Xinje XDPPro project, PLC1: XD3-32 (software 3.7.14 2021-12-24)

PROGRAM 梯形图

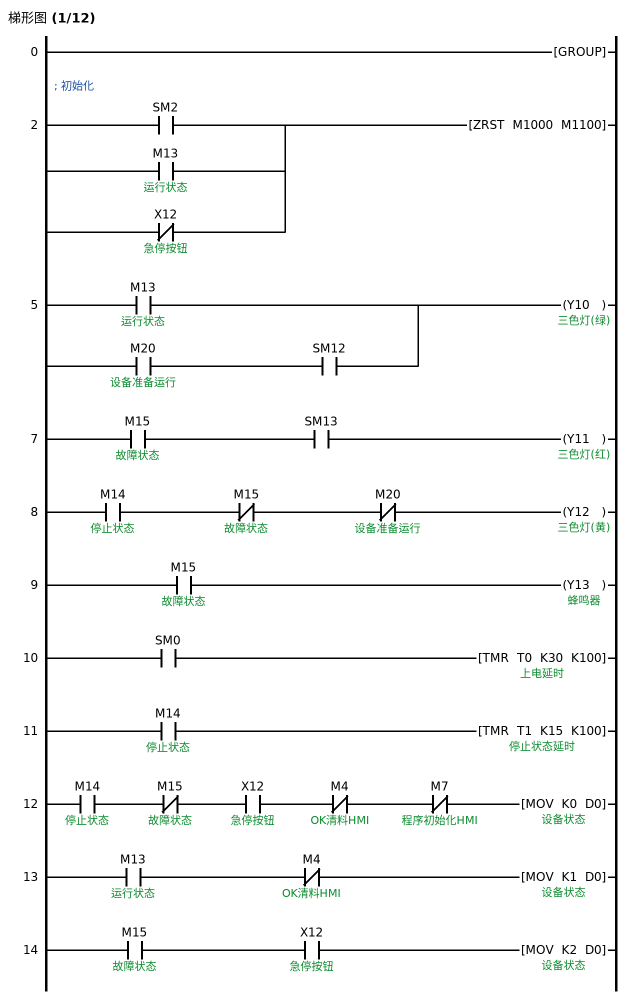
GROUP
; 初始化
LD     SM2
OR     M13	; 运行状态
ORI    X12	; 急停按钮
ZRST   M1000 M1100
LD     M13	; 运行状态
LD     M20	; 设备准备运行
AND    SM12
ORB
OUT    Y10	; 三色灯(绿)
LD     M15	; 故障状态
AND    SM13
OUT    Y11	; 三色灯(红)
LD     M14	; 停止状态
ANI    M15	; 故障状态
ANI    M20	; 设备准备运行
OUT    Y12	; 三色灯(黄)
LD     M15	; 故障状态
OUT    Y13	; 蜂鸣器
LD     SM0
TMR    T0 K30 K100	; 上电延时
LD     M14	; 停止状态
TMR    T1 K15 K100	; 停止状态延时
LD     M14	; 停止状态
ANI    M15	; 故障状态
AND    X12	; 急停按钮
ANI    M4	; OK清料HMI
ANI    M7	; 程序初始化HMI
MOV    K0 D0	; 设备状态
LD     M13	; 运行状态
ANI    M4	; OK清料HMI
MOV    K1 D0	; 设备状态
LD     M15	; 故障状态
AND    X12	; 急停按钮
MOV    K2 D0	; 设备状态

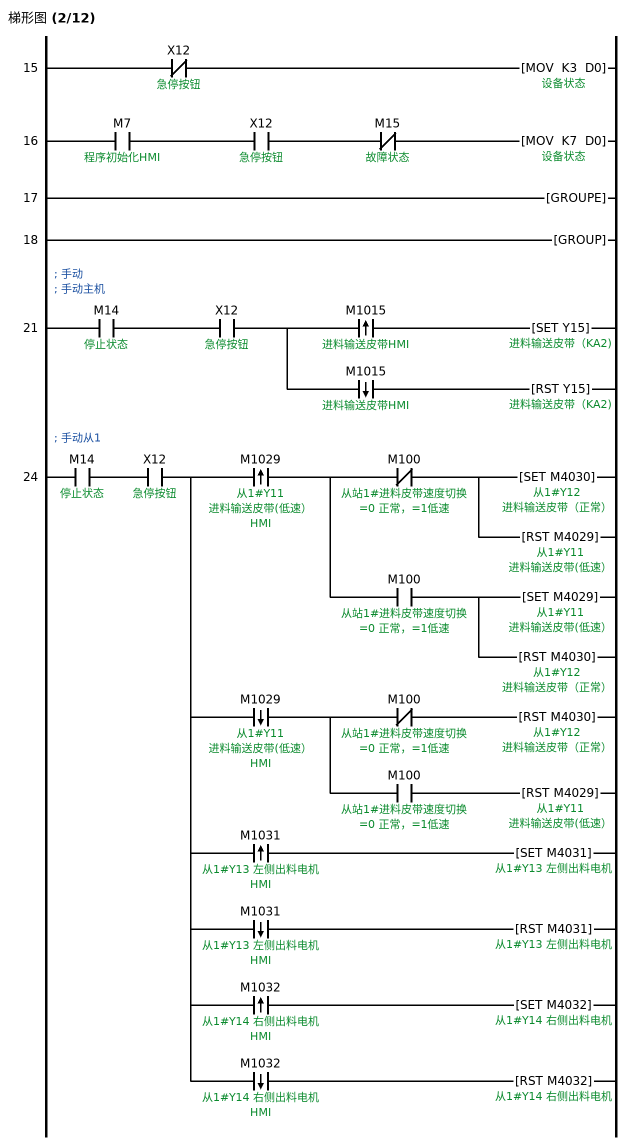
LDI    X12	; 急停按钮
MOV    K3 D0	; 设备状态
LD     M7	; 程序初始化HMI
AND    X12	; 急停按钮
ANI    M15	; 故障状态
MOV    K7 D0	; 设备状态
GROUPE
GROUP
; 手动
; 手动主机
LD     M14	; 停止状态
AND    X12	; 急停按钮
MPS
ANDP   M1015	; 进料输送皮带HMI
SET    Y15	; 进料输送皮带（KA2)
MPP
ANDF   M1015	; 进料输送皮带HMI
RST    Y15	; 进料输送皮带（KA2)
; 手动从1
LD     M14	; 停止状态
AND    X12	; 急停按钮
MPS
ANDP   M1029	; 从1#Y11 进料输送皮带(低速）       HMI
MPS
ANI    M100	; 从站1#进料皮带速度切换=0 正常，=1低速
SET    M4030	; 从1#Y12 进料输送皮带（正常）
RST    M4029	; 从1#Y11 进料输送皮带(低速）
MPP
AND    M100	; 从站1#进料皮带速度切换=0 正常，=1低速
SET    M4029	; 从1#Y11 进料输送皮带(低速）
RST    M4030	; 从1#Y12 进料输送皮带（正常）
MRD
ANDF   M1029	; 从1#Y11 进料输送皮带(低速）       HMI
MPS
ANI    M100	; 从站1#进料皮带速度切换=0 正常，=1低速
RST    M4030	; 从1#Y12 进料输送皮带（正常）
MPP
AND    M100	; 从站1#进料皮带速度切换=0 正常，=1低速
RST    M4029	; 从1#Y11 进料输送皮带(低速）
MRD
ANDP   M1031	; 从1#Y13 左侧出料电机       HMI
SET    M4031	; 从1#Y13 左侧出料电机
MRD
ANDF   M1031	; 从1#Y13 左侧出料电机       HMI
RST    M4031	; 从1#Y13 左侧出料电机
MRD
ANDP   M1032	; 从1#Y14 右侧出料电机       HMI
SET    M4032	; 从1#Y14 右侧出料电机
MPP
ANDF   M1032	; 从1#Y14 右侧出料电机       HMI
RST    M4032	; 从1#Y14 右侧出料电机

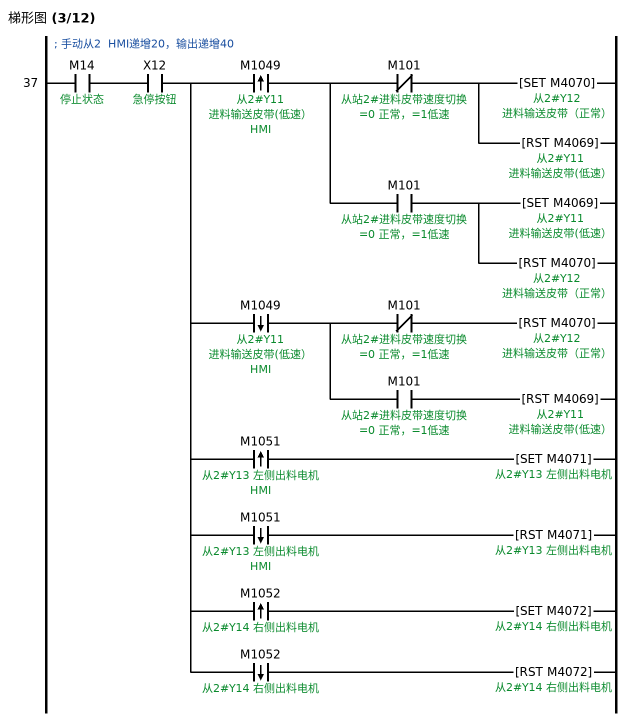
; 手动从2  HMI递增20，输出递增40
LD     M14	; 停止状态
AND    X12	; 急停按钮
MPS
ANDP   M1049	; 从2#Y11 进料输送皮带(低速）       HMI
MPS
ANI    M101	; 从站2#进料皮带速度切换=0 正常，=1低速
SET    M4070	; 从2#Y12 进料输送皮带（正常）
RST    M4069	; 从2#Y11 进料输送皮带(低速）
MPP
AND    M101	; 从站2#进料皮带速度切换=0 正常，=1低速
SET    M4069	; 从2#Y11 进料输送皮带(低速）
RST    M4070	; 从2#Y12 进料输送皮带（正常）
MRD
ANDF   M1049	; 从2#Y11 进料输送皮带(低速）       HMI
MPS
ANI    M101	; 从站2#进料皮带速度切换=0 正常，=1低速
RST    M4070	; 从2#Y12 进料输送皮带（正常）
MPP
AND    M101	; 从站2#进料皮带速度切换=0 正常，=1低速
RST    M4069	; 从2#Y11 进料输送皮带(低速）
MRD
ANDP   M1051	; 从2#Y13 左侧出料电机       HMI
SET    M4071	; 从2#Y13 左侧出料电机
MRD
ANDF   M1051	; 从2#Y13 左侧出料电机       HMI
RST    M4071	; 从2#Y13 左侧出料电机
MRD
ANDP   M1052	; 从2#Y14 右侧出料电机
SET    M4072	; 从2#Y14 右侧出料电机
MPP
ANDF   M1052	; 从2#Y14 右侧出料电机
RST    M4072	; 从2#Y14 右侧出料电机

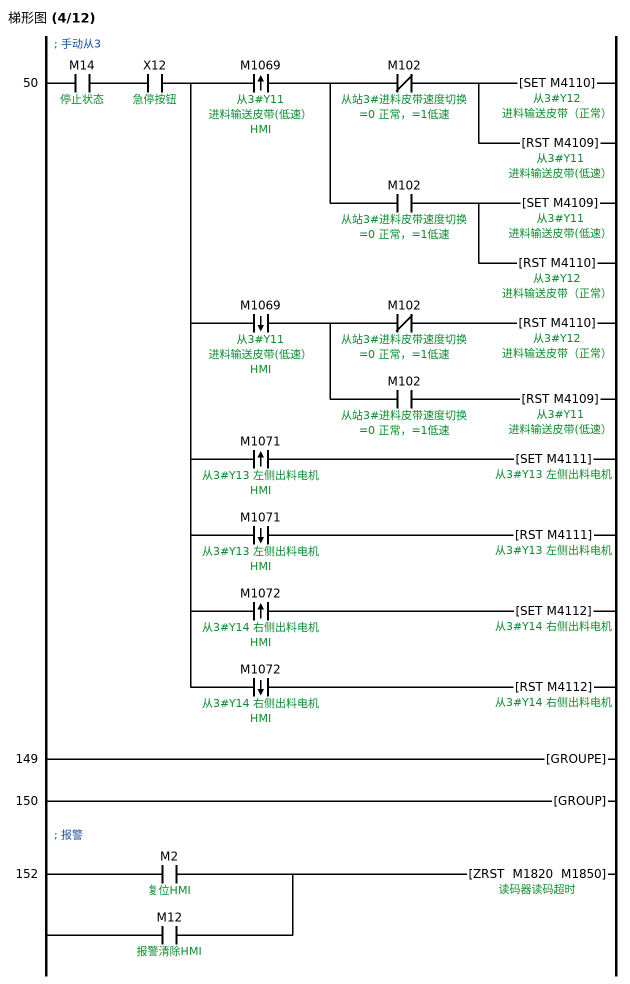
; 手动从3
LD     M14	; 停止状态
AND    X12	; 急停按钮
MPS
ANDP   M1069	; 从3#Y11 进料输送皮带(低速）       HMI
MPS
ANI    M102	; 从站3#进料皮带速度切换=0 正常，=1低速
SET    M4110	; 从3#Y12 进料输送皮带（正常）
RST    M4109	; 从3#Y11 进料输送皮带(低速）
MPP
AND    M102	; 从站3#进料皮带速度切换=0 正常，=1低速
SET    M4109	; 从3#Y11 进料输送皮带(低速）
RST    M4110	; 从3#Y12 进料输送皮带（正常）
MRD
ANDF   M1069	; 从3#Y11 进料输送皮带(低速）       HMI
MPS
ANI    M102	; 从站3#进料皮带速度切换=0 正常，=1低速
RST    M4110	; 从3#Y12 进料输送皮带（正常）
MPP
AND    M102	; 从站3#进料皮带速度切换=0 正常，=1低速
RST    M4109	; 从3#Y11 进料输送皮带(低速）
MRD
ANDP   M1071	; 从3#Y13 左侧出料电机       HMI
SET    M4111	; 从3#Y13 左侧出料电机
MRD
ANDF   M1071	; 从3#Y13 左侧出料电机       HMI
RST    M4111	; 从3#Y13 左侧出料电机
MRD
ANDP   M1072	; 从3#Y14 右侧出料电机       HMI
SET    M4112	; 从3#Y14 右侧出料电机
MPP
ANDF   M1072	; 从3#Y14 右侧出料电机       HMI
RST    M4112	; 从3#Y14 右侧出料电机
GROUPE
GROUP
; 报警
LD     M2	; 复位HMI
OR     M12	; 报警清除HMI
ZRST   M1820 M1850	; 读码器读码超时

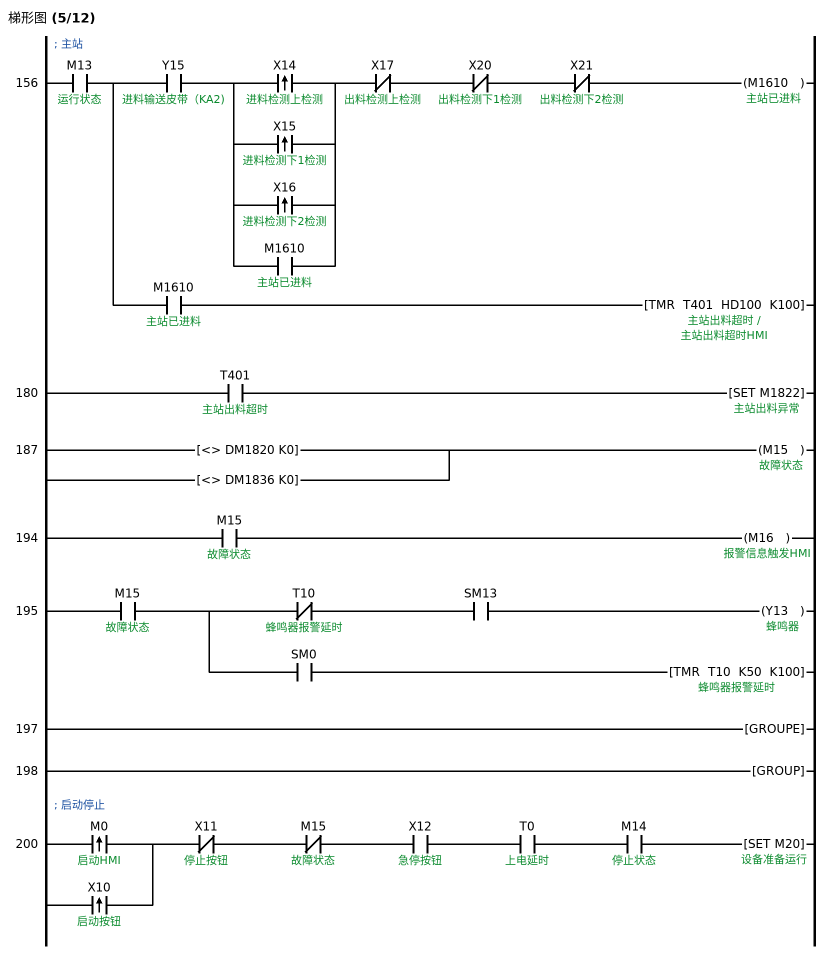
; 主站
LD     M13	; 运行状态
MPS
AND    Y15	; 进料输送皮带（KA2)
LDP    X14	; 进料检测上检测
ORP    X15	; 进料检测下1检测
ORP    X16	; 进料检测下2检测
OR     M1610	; 主站已进料
ANB
ANI    X17	; 出料检测上检测
ANI    X20	; 出料检测下1检测
ANI    X21	; 出料检测下2检测
OUT    M1610	; 主站已进料
MPP
AND    M1610	; 主站已进料
TMR    T401 HD100 K100	; 主站出料超时 / 主站出料超时HMI
LD     T401	; 主站出料超时
SET    M1822	; 主站出料异常
LD<>   DM1820 K0
OR<>   DM1836 K0
OUT    M15	; 故障状态
LD     M15	; 故障状态
OUT    M16	; 报警信息触发HMI
LD     M15	; 故障状态
MPS
ANI    T10	; 蜂鸣器报警延时
AND    SM13
OUT    Y13	; 蜂鸣器
MPP
AND    SM0
TMR    T10 K50 K100	; 蜂鸣器报警延时
GROUPE
GROUP
; 启动停止
LDP    M0	; 启动HMI
ORP    X10	; 启动按钮
ANI    X11	; 停止按钮
ANI    M15	; 故障状态
AND    X12	; 急停按钮
AND    T0	; 上电延时
AND    M14	; 停止状态
SET    M20	; 设备准备运行

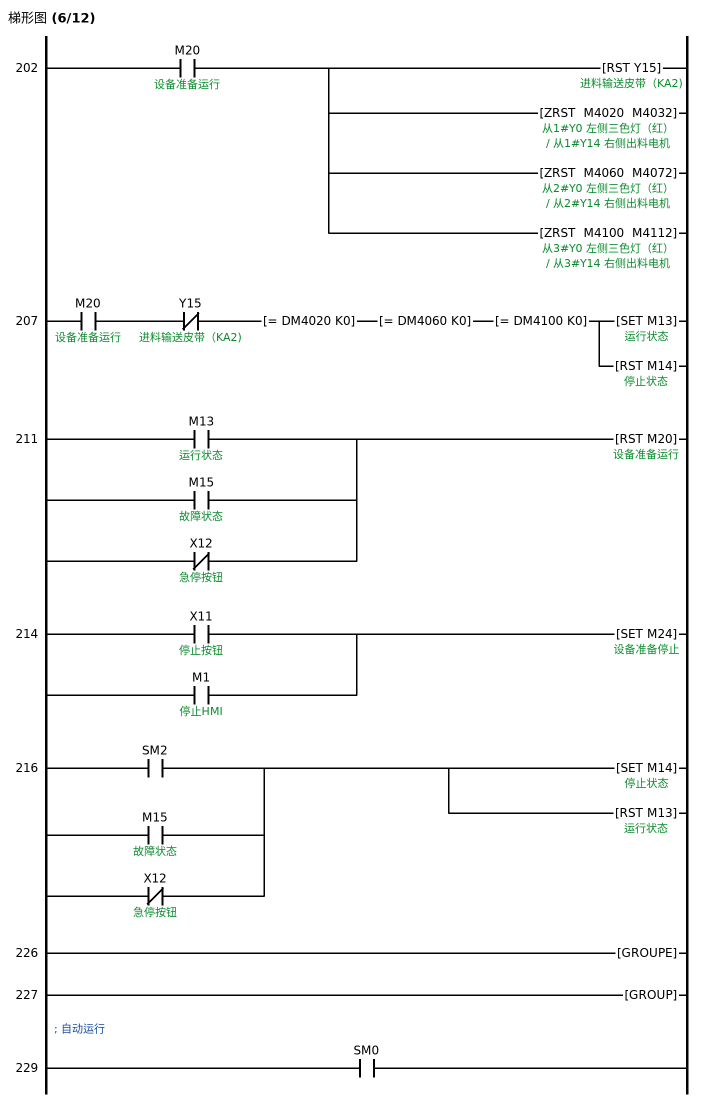
LD     M20	; 设备准备运行
RST    Y15	; 进料输送皮带（KA2)
ZRST   M4020 M4032	; 从1#Y0 左侧三色灯（红） / 从1#Y14 右侧出料电机
ZRST   M4060 M4072	; 从2#Y0 左侧三色灯（红） / 从2#Y14 右侧出料电机
ZRST   M4100 M4112	; 从3#Y0 左侧三色灯（红） / 从3#Y14 右侧出料电机
LD     M20	; 设备准备运行
ANI    Y15	; 进料输送皮带（KA2)
AND=   DM4020 K0
AND=   DM4060 K0
AND=   DM4100 K0
SET    M13	; 运行状态
RST    M14	; 停止状态
LD     M13	; 运行状态
OR     M15	; 故障状态
ORI    X12	; 急停按钮
RST    M20	; 设备准备运行
LD     X11	; 停止按钮
OR     M1	; 停止HMI
SET    M24	; 设备准备停止
LD     SM2
OR     M15	; 故障状态
ORI    X12	; 急停按钮
SET    M14	; 停止状态
RST    M13	; 运行状态
GROUPE
GROUP
; 自动运行
LD     SM0

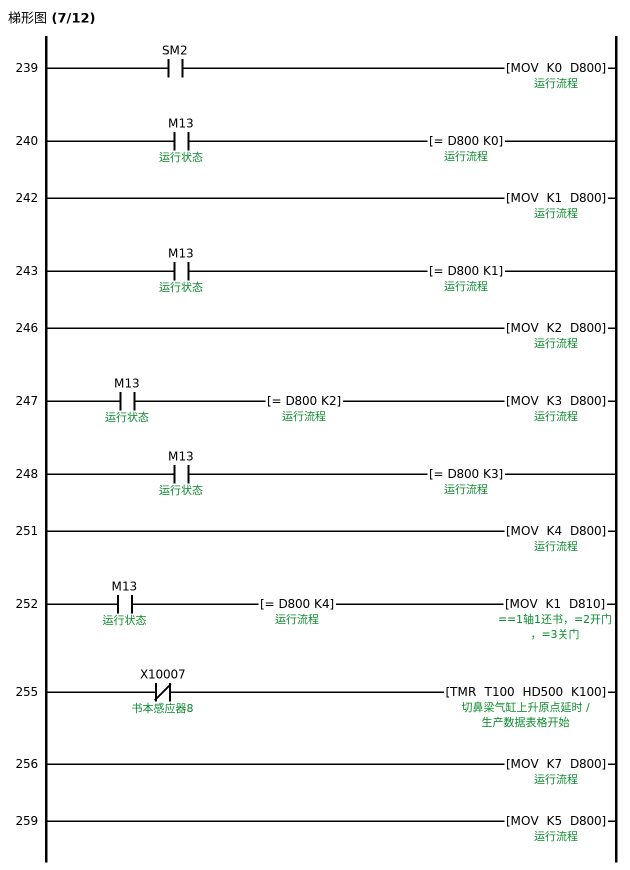
LD     SM2
MOV    K0 D800	; 运行流程
LD     M13	; 运行状态
AND=   D800 K0	; 运行流程
MOV    K1 D800	; 运行流程
LD     M13	; 运行状态
AND=   D800 K1	; 运行流程
MOV    K2 D800	; 运行流程
LD     M13	; 运行状态
AND=   D800 K2	; 运行流程
MOV    K3 D800	; 运行流程
LD     M13	; 运行状态
AND=   D800 K3	; 运行流程
MOV    K4 D800	; 运行流程
LD     M13	; 运行状态
AND=   D800 K4	; 运行流程
MOV    K1 D810	; ==1轴1还书，=2开门，=3关门
LDI    X10007	; 书本感应器8
TMR    T100 HD500 K100	; 切鼻梁气缸上升原点延时 / 生产数据表格开始
MOV    K7 D800	; 运行流程
MOV    K5 D800	; 运行流程

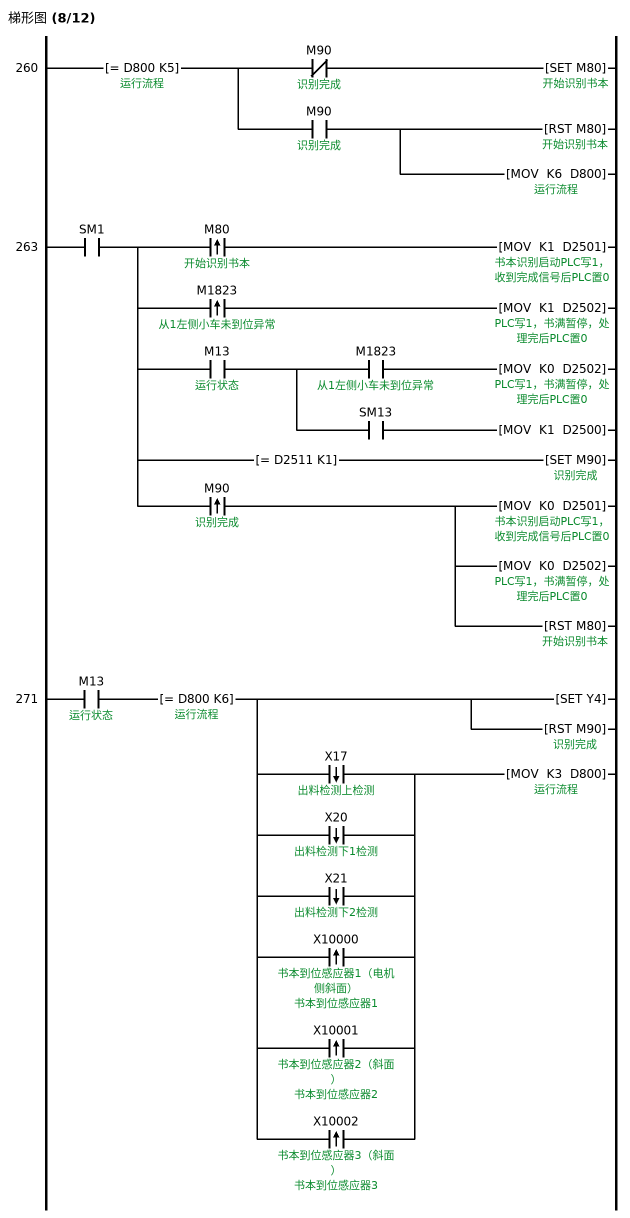
LD=    D800 K5	; 运行流程
MPS
ANI    M90	; 识别完成
SET    M80	; 开始识别书本
MPP
AND    M90	; 识别完成
RST    M80	; 开始识别书本
MOV    K6 D800	; 运行流程
LD     SM1
MPS
ANDP   M80	; 开始识别书本
MOV    K1 D2501	; 书本识别启动PLC写1，收到完成信号后PLC置0
MRD
ANDP   M1823	; 从1左侧小车未到位异常
MOV    K1 D2502	; PLC写1，书满暂停，处理完后PLC置0
MRD
AND    M13	; 运行状态
MPS
AND    M1823	; 从1左侧小车未到位异常
MOV    K0 D2502	; PLC写1，书满暂停，处理完后PLC置0
MPP
AND    SM13
MOV    K1 D2500
MRD
AND=   D2511 K1
SET    M90	; 识别完成
MPP
ANDP   M90	; 识别完成
MOV    K0 D2501	; 书本识别启动PLC写1，收到完成信号后PLC置0
MOV    K0 D2502	; PLC写1，书满暂停，处理完后PLC置0
RST    M80	; 开始识别书本
LD     M13	; 运行状态
AND=   D800 K6	; 运行流程
SET    Y4
RST    M90	; 识别完成
LDF    X17	; 出料检测上检测
ORF    X20	; 出料检测下1检测
ORF    X21	; 出料检测下2检测
ORP    X10000	; 书本到位感应器1（电机侧斜面）       书本到位感应器1
ORP    X10001	; 书本到位感应器2（斜面）             书本到位感应器2
ORP    X10002	; 书本到位感应器3（斜面）             书本到位感应器3
ANB
MOV    K3 D800	; 运行流程

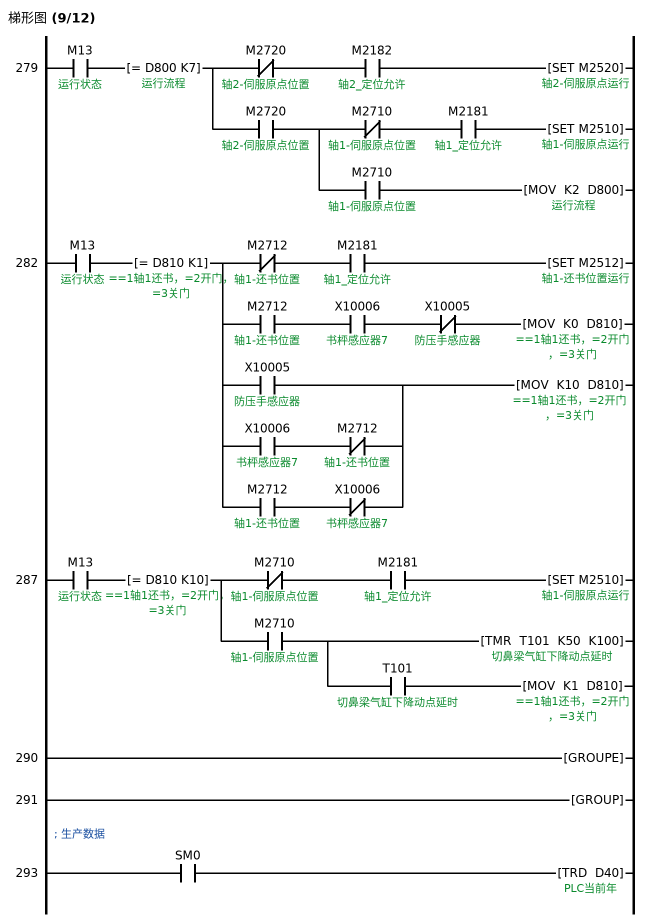
LD     M13	; 运行状态
AND=   D800 K7	; 运行流程
MPS
ANI    M2720	; 轴2-伺服原点位置
AND    M2182	; 轴2_定位允许
SET    M2520	; 轴2-伺服原点运行
MPP
AND    M2720	; 轴2-伺服原点位置
MPS
ANI    M2710	; 轴1-伺服原点位置
AND    M2181	; 轴1_定位允许
SET    M2510	; 轴1-伺服原点运行
MPP
AND    M2710	; 轴1-伺服原点位置
MOV    K2 D800	; 运行流程
LD     M13	; 运行状态
AND=   D810 K1	; ==1轴1还书，=2开门，=3关门
MPS
ANI    M2712	; 轴1-还书位置
AND    M2181	; 轴1_定位允许
SET    M2512	; 轴1-还书位置运行
MRD
AND    M2712	; 轴1-还书位置
AND    X10006	; 书枰感应器7
ANI    X10005	; 防压手感应器
MOV    K0 D810	; ==1轴1还书，=2开门，=3关门
MPP
LD     X10005	; 防压手感应器
LD     X10006	; 书枰感应器7
ANI    M2712	; 轴1-还书位置
ORB
LD     M2712	; 轴1-还书位置
ANI    X10006	; 书枰感应器7
ORB
ANB
MOV    K10 D810	; ==1轴1还书，=2开门，=3关门
LD     M13	; 运行状态
AND=   D810 K10	; ==1轴1还书，=2开门，=3关门
MPS
ANI    M2710	; 轴1-伺服原点位置
AND    M2181	; 轴1_定位允许
SET    M2510	; 轴1-伺服原点运行
MPP
AND    M2710	; 轴1-伺服原点位置
TMR    T101 K50 K100	; 切鼻梁气缸下降动点延时
AND    T101	; 切鼻梁气缸下降动点延时
MOV    K1 D810	; ==1轴1还书，=2开门，=3关门
GROUPE
GROUP
; 生产数据
LD     SM0
TRD    D40	; PLC当前年

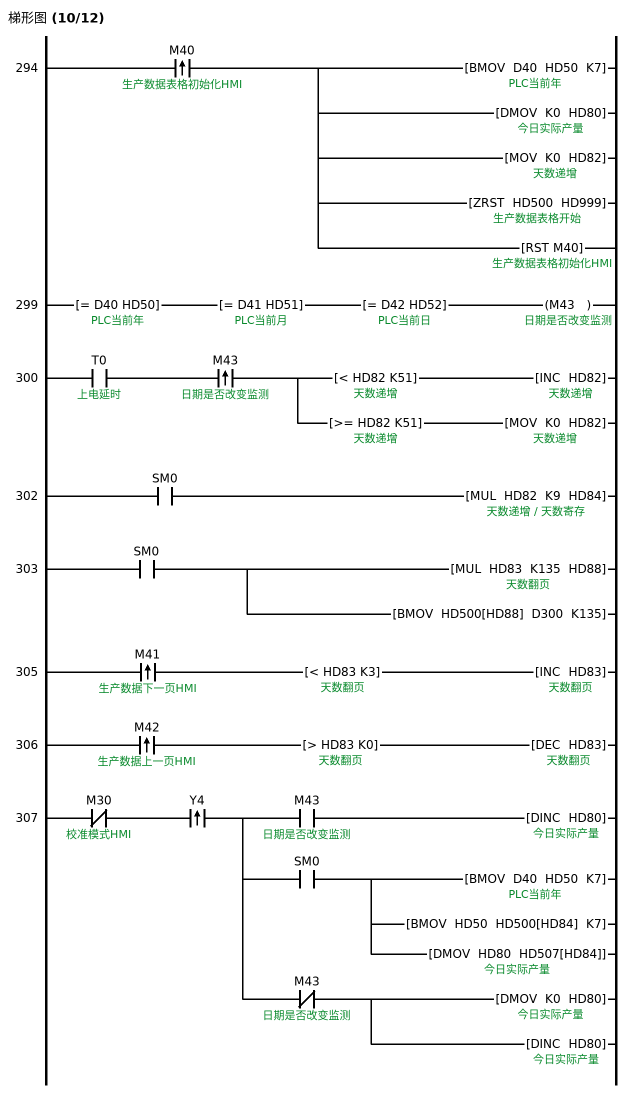
LDP    M40	; 生产数据表格初始化HMI
BMOV   D40 HD50 K7	; PLC当前年
DMOV   K0 HD80	; 今日实际产量
MOV    K0 HD82	; 天数递增
ZRST   HD500 HD999	; 生产数据表格开始
RST    M40	; 生产数据表格初始化HMI
LD=    D40 HD50	; PLC当前年
AND=   D41 HD51	; PLC当前月
AND=   D42 HD52	; PLC当前日
OUT    M43	; 日期是否改变监测
LD     T0	; 上电延时
ANDP   M43	; 日期是否改变监测
MPS
AND<   HD82 K51	; 天数递增
INC    HD82	; 天数递增
MPP
AND>=  HD82 K51	; 天数递增
MOV    K0 HD82	; 天数递增
LD     SM0
MUL    HD82 K9 HD84	; 天数递增 / 天数寄存
LD     SM0
MUL    HD83 K135 HD88	; 天数翻页
BMOV   HD500[HD88] D300 K135
LDP    M41	; 生产数据下一页HMI
AND<   HD83 K3	; 天数翻页
INC    HD83	; 天数翻页
LDP    M42	; 生产数据上一页HMI
AND>   HD83 K0	; 天数翻页
DEC    HD83	; 天数翻页
LDI    M30	; 校准模式HMI
ANDP   Y4
MPS
AND    M43	; 日期是否改变监测
DINC   HD80	; 今日实际产量
MRD
AND    SM0
BMOV   D40 HD50 K7	; PLC当前年
BMOV   HD50 HD500[HD84] K7
DMOV   HD80 HD507[HD84]	; 今日实际产量
MPP
ANI    M43	; 日期是否改变监测
DMOV   K0 HD80	; 今日实际产量
DINC   HD80	; 今日实际产量

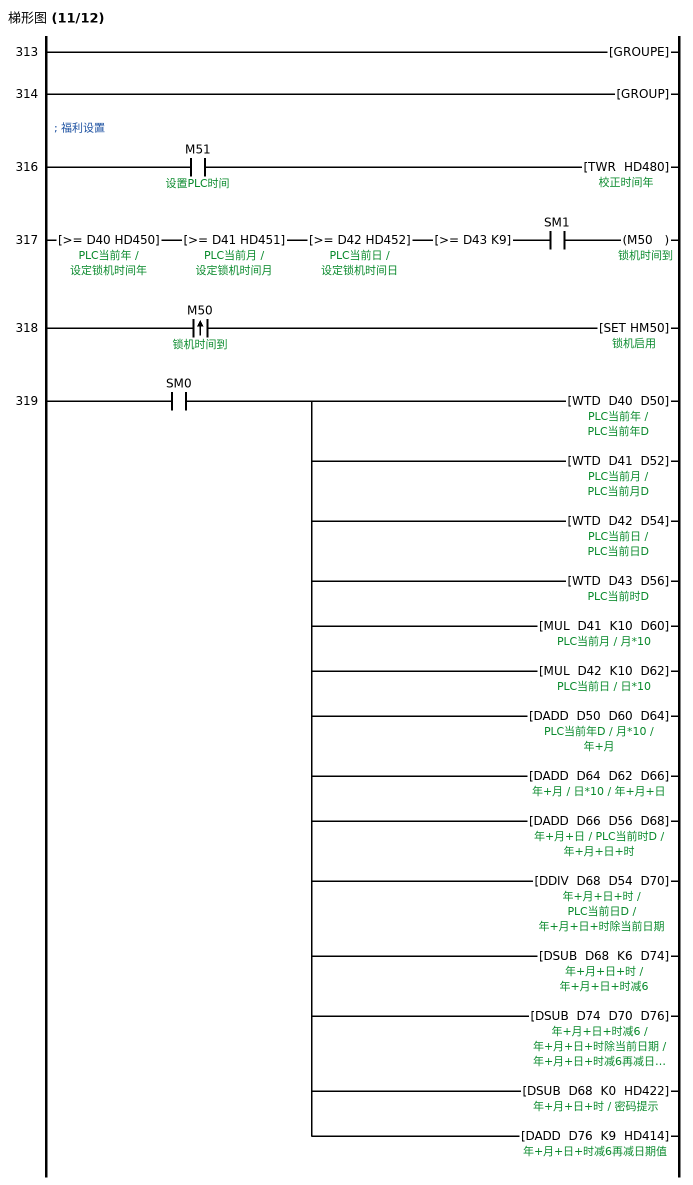
GROUPE
GROUP
; 福利设置
LD     M51	; 设置PLC时间
TWR    HD480	; 校正时间年
LD>=   D40 HD450	; PLC当前年 / 设定锁机时间年
AND>=  D41 HD451	; PLC当前月 / 设定锁机时间月
AND>=  D42 HD452	; PLC当前日 / 设定锁机时间日
AND>=  D43 K9
AND    SM1
OUT    M50	; 锁机时间到
LDP    M50	; 锁机时间到
SET    HM50	; 锁机启用
LD     SM0
WTD    D40 D50	; PLC当前年 / PLC当前年D
WTD    D41 D52	; PLC当前月 / PLC当前月D
WTD    D42 D54	; PLC当前日 / PLC当前日D
WTD    D43 D56	; PLC当前时D
MUL    D41 K10 D60	; PLC当前月 / 月*10
MUL    D42 K10 D62	; PLC当前日 / 日*10
DADD   D50 D60 D64	; PLC当前年D / 月*10 / 年+月
DADD   D64 D62 D66	; 年+月 / 日*10 / 年+月+日
DADD   D66 D56 D68	; 年+月+日 / PLC当前时D / 年+月+日+时
DDIV   D68 D54 D70	; 年+月+日+时 / PLC当前日D / 年+月+日+时除当前日期
DSUB   D68 K6 D74	; 年+月+日+时 / 年+月+日+时减6
DSUB   D74 D70 D76	; 年+月+日+时减6 / 年+月+日+时除当前日期 / 年+月+日+时减6再减日期值
DSUB   D68 K0 HD422	; 年+月+日+时 / 密码提示
DADD   D76 K9 HD414	; 年+月+日+时减6再减日期值

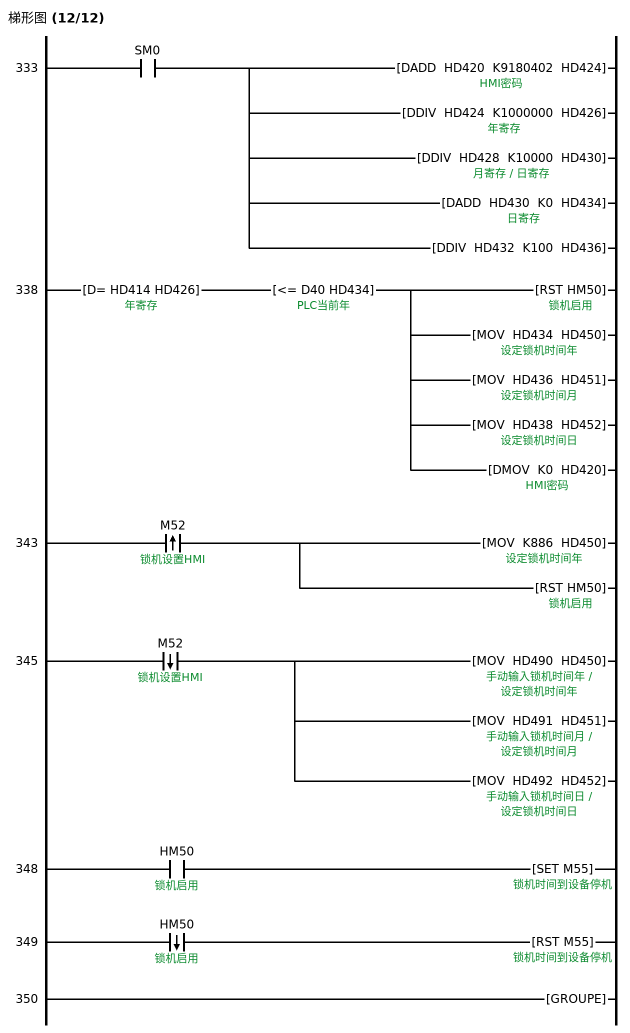
LD     SM0
DADD   HD420 K9180402 HD424	; HMI密码
DDIV   HD424 K1000000 HD426	; 年寄存
DDIV   HD428 K10000 HD430	; 月寄存 / 日寄存
DADD   HD430 K0 HD434	; 日寄存
DDIV   HD432 K100 HD436
DLD=   HD414 HD426	; 年寄存
AND<=  D40 HD434	; PLC当前年
RST    HM50	; 锁机启用
MOV    HD434 HD450	; 设定锁机时间年
MOV    HD436 HD451	; 设定锁机时间月
MOV    HD438 HD452	; 设定锁机时间日
DMOV   K0 HD420	; HMI密码
LDP    M52	; 锁机设置HMI
MOV    K886 HD450	; 设定锁机时间年
RST    HM50	; 锁机启用
LDF    M52	; 锁机设置HMI
MOV    HD490 HD450	; 手动输入锁机时间年 / 设定锁机时间年
MOV    HD491 HD451	; 手动输入锁机时间月 / 设定锁机时间月
MOV    HD492 HD452	; 手动输入锁机时间日 / 设定锁机时间日
LD     HM50	; 锁机启用
SET    M55	; 锁机时间到设备停机
LDF    HM50	; 锁机启用
RST    M55	; 锁机时间到设备停机
GROUPE

COMMENTS (devices not used above)
M3	急停HMI
M5	NG清料HMI
M6	轴复位HMI
M8	参数默认HMI
M9	产量清零HMI
M10	当前产量清零HMI
M21	軸总復位中
M22	设备复位中
M25	设备清料完成
M2042	轴2_JOG快慢速HMI
M2021	轴1_JOG- HMI
M2022	轴2_JOG- HMI
M2041	轴1_JOG快慢速HMI
M2002	轴2_JOG+ HMI
M1821	与读码器通信异常
HD200	轴2_JOG快速度HMI
HD202	轴2_JOG慢速度HMI
HD204	轴2_JOG速度寄存
HD206	轴2_JOG增量
HD208	轴2_JOG位置寄存
HD210	轴2_回零速度
HD212	轴2_运行速度HMI
HD214	轴2_自动加速度
HD215	轴2_自动减速度
HD218	轴2_定位位置寄存
D2100	轴1_JOG快速度
D2102	轴1_JOG慢速度
D2104	轴1_JOG速度寄存
D2106	轴1_JOG增量
D2108	轴1_JOG位置寄存
D2110	轴1_回零速度
D2112	轴1_运行速度
D2114	轴1_自动加速度
D2115	轴1_自动减速度
D2116	轴1_JOG加速度
D2117	轴1_JOG减速度
D2118	轴1_定位位置寄存
HD216	轴2_手动加速度
HD217	轴2_手动减速度
M2141	轴1_伺服回零中
M1200	快慢速切换HMI
M1020	从1#Y0 左侧三色灯（红）       HMI
HD8	切鼻梁个数计数
HD220	轴2_鼻梁长度设置HMI
HD12	滚刀切料个数计数
M2001	轴1_JOG+ HMI
HD40	Y0当前脉冲值记忆
HD42	Y1当前脉冲值记忆
T2	超声波休眠延时
HD2	超声波休眠时间
T3	超声运行延时
HD300	生产速度HMI
HD310	鼻梁滚轮周长HMI
HD102	轴1_JOG慢速度HMI
HD104	轴1_JOG速度寄存
HD106	轴1_JOG增量
HD108	轴1_JOG位置寄存
HD110	轴1_回零速度
HD112	轴1_运行速度HMI
HD114	轴1_自动加速度
HD115	轴1_自动减速度
HD116	轴1_JOG加速度
HD117	轴1_JOG减速度
HD118	轴1_定位位置寄存
D108	鼻梁长度计算脉冲结果
D100	K750浮点数
D104	鼻梁长度计算脉冲结果寄存
D142	输出脉冲频率浮点数
HD32	生产效率寄存2
HD20	设定产量HMI
HD22	实际产量(切鼻梁个数计数)
HD30	生产效率寄存1
M1600	产量达成
HM30	内置鼻梁标志/外置鼻梁HMI
HD24	滚刀切料个数计数
HD34	生产效率
HM32	校准完成
M1826	从1右侧小车未到位异常
HM3	急停后切断鼻梁
M1827	从1右侧料满异常
M18	手动操作记忆标志
HD507	当日实际产量
HD400	当前时间年
HD401	当前时间月
HD402	当前时间日
HD403	当前时间时
HD453	设定锁机时间时
HD481	校正时间月
HD482	校正时间日
HD483	校正时间时
D72	年+月+日+时除当前日期得商
HD28	累计产量
X10003	小车感应光栅
X10004	小车到位感应（对射）
M2101	轴1_伺服回零HMI
M2102	轴2_伺服回零HMI
M2121	轴1_伺服回零允许
M2122	轴2_伺服回零允许
M2142	轴2_伺服回零中
M2161	轴1_原点确定
M2162	轴2_原点确定
M2201	轴1_JOG连续/增量HMI
M2202	轴2_JOG连续/增量HMI
M2241	轴1_增量JOG运行
M2242	轴2_增量JOG运行
M2310	轴1-伺服原点运行HMI
M2311	轴1-伺服定位运行HMI
M2320	轴2-伺服原点运行HMI
M2321	轴2-伺服定位运行HMI
M2511	轴1-伺服定位运行
M2521	轴2-伺服定位运行
M2711	轴1-伺服定位位置
M2721	轴2-伺服定位位置
HD894	轴1_设置每次回零计数HMI
HD895	轴1_当前每次回零计数
HD900	轴2_JOG快速度HMI
HD902	轴2_JOG慢速度HMI
HD904	轴2_JOG速度寄存
HD906	轴2_JOG增量
HD908	轴2_JOG位置寄存
HD910	轴2_回零速度
HD912	轴2_运行速度HMI
HD914	轴2_自动加速度
HD915	轴2_自动减速度
HD916	轴2_手动加速度
HD917	轴2_手动减速度
HD918	轴2_定位位置寄存
HD920	轴2__原点位置HMI
HD922	轴2__定位位置HMI
HD994	轴2_设置每次回零计数HMI
HD995	轴2_当前每次回零计数
HD800	轴1_JOG快速度HMI
HD802	轴1_JOG慢速度HMI
HD804	轴1_JOG速度寄存
HD806	轴1_JOG增量
HD808	轴1_JOG位置寄存
HD810	轴1_回零速度
HD812	轴1_运行速度HMI
HD814	轴1_自动加速度
HD815	轴1_自动减速度
HD816	轴1_JOG加速度
HD817	轴1_JOG减速度
HD818	轴1_定位位置寄存
HD820	轴1__原点位置HMI
HD822	轴1__定位位置HMI
D851	轴1-回原点流程
HD890	轴1-正软限位HMI
HD892	轴1-负软限位HMI
T422	轴1 启动
HD888	轴1—当前脉冲数
HD988	轴2当前脉冲数
M1021	从1#Y1 左侧三色灯（绿）       HMI
M1828	从1右侧出料异常
D852	轴2-回原流程
T424	轴2定位允许
M1825	从1左侧出料异常
M2312	还书位置运行-HMI
M1824	从1左侧料满异常
M1022	从1#Y2 左侧三色灯（黄）       HMI
M1023	从1#Y3 右侧三色灯（红）       HMI
M1024	从1#Y4 右侧三色灯（绿）       HMI
M1025	从1#Y5 右侧三色灯（黄）       HMI
M1026	从1#Y6 出料三色灯（红）       HMI
M1027	从1#Y7 出料三色灯（绿）       HMI
M1028	从1#Y10 出料三色灯（黄）       HMI
M1030	从1#Y12 进料输送皮带（正常）       HMI
M1040	从2#Y0 左侧三色灯（红）       HMI
M1041	从2#Y1 左侧三色灯（绿）       HMI
M1042	从2#Y2 左侧三色灯（黄）       HMI
M1043	从2#Y3 右侧三色灯（红）       HMI
M1044	从2#Y4 右侧三色灯（绿）       HMI
M1045	从2#Y5 右侧三色灯（黄）       HMI
M1046	从2#Y6 出料三色灯（红）       HMI
M1047	从2#Y7 出料三色灯（绿）       HMI
M1048	从2#Y10 出料三色灯（黄）       HMI
M1050	从2#Y12 进料输送皮带（正常）       HMI
M1060	从3#Y0 左侧三色灯（红）       HMI
M1061	从3#Y1 左侧三色灯（绿）       HMI
M1062	从3#Y2 左侧三色灯（黄）       HMI
M1063	从3#Y3 右侧三色灯（红）       HMI
M1064	从3#Y4 右侧三色灯（绿）       HMI
M1065	从3#Y5 右侧三色灯（黄）       HMI
M1066	从3#Y6 出料三色灯（红）       HMI
M1067	从3#Y7 出料三色灯（绿）       HMI
M1068	从3#Y10 出料三色灯（黄）       HMI
M1070	从3#Y12 进料输送皮带（正常）       HMI
M4000	从1#X0进料检测上检测
M4001	从1#X1进料检测下1检测
M4002	从1#X2进料检测下2检测
M4003	从1#X3左侧出料上检测
M4004	从1#X4左侧出料下1检测
M4005	从1#X5左侧出料下2检测
M4006	从1#X6左侧料箱检测
M4007	从1#X7左侧料箱满料检测
M4008	从1#X10右侧出料上检测
M4009	从1#X11右侧出料下1检测
M4010	从1#X12右侧出料下2检测
M4011	从1#X13右侧料箱检测
M4012	从1#X14右侧料箱满料检测
M4013	从1#X15出料检测上检测
M4014	从1#X16出料检测下1检测
M4015	从1#X17出料检测下2检测
M4021	从1#Y1 左侧三色灯（绿）
M4022	从1#Y2 左侧三色灯（黄）
M4023	从1#Y3 右侧三色灯（红）
M4024	从1#Y4 右侧三色灯（绿）
M4025	从1#Y5 右侧三色灯（黄）
M4026	从1#Y6 出料三色灯（红）
M4027	从1#Y7 出料三色灯（绿）
M4028	从1#Y10 出料三色灯（黄）
M4040	从2#X0进料检测上检测
M4041	从2#X1进料检测下1检测
M4042	从2#X2进料检测下2检测
M4043	从2#X3左侧出料上检测
M4044	从2#X4左侧出料下1检测
M4045	从2#X5左侧出料下2检测
M4046	从2#X6左侧料箱检测
M4047	从2#X7左侧料箱满料检测
M4048	从2#X10右侧出料上检测
M4049	从2#X11右侧出料下1检测
M4050	从2#X12右侧出料下2检测
M4051	从2#X13右侧料箱检测
M4052	从2#X14右侧料箱满料检测
M4053	从2#X15出料检测上检测
M4054	从2#X16出料检测下1检测
M4055	从2#X17出料检测下2检测
M4061	从2#Y1 左侧三色灯（绿）
M4062	从2#Y2 左侧三色灯（黄）
M4063	从2#Y3 右侧三色灯（红）
M4064	从2#Y4 右侧三色灯（绿）
M4065	从2#Y5 右侧三色灯（黄）
M4066	从2#Y6 出料三色灯（红）
M4067	从2#Y7 出料三色灯（绿）
M4068	从2#Y10 出料三色灯（黄）
M4080	从3#X0进料检测上检测
M4081	从3#X1进料检测下1检测
M4082	从3#X2进料检测下2检测
M4083	从3#X3左侧出料上检测
M4084	从3#X4左侧出料下1检测
M4085	从3#X5左侧出料下2检测
M4086	从3#X6左侧料箱检测
M4087	从3#X7左侧料箱满料检测
M4088	从3#X10右侧出料上检测
M4089	从3#X11右侧出料下1检测
M4090	从3#X12右侧出料下2检测
M4091	从3#X13右侧料箱检测
M4092	从3#X14右侧料箱满料检测
M4093	从3#X15出料检测上检测
M4094	从3#X16出料检测下1检测
M4095	从3#X17出料检测下2检测
M4096	从3#X20出料箱检测
M4097	从3#X21出料箱满料检测
M4101	从3#Y1 左侧三色灯（绿）
M4102	从3#Y2 左侧三色灯（黄）
M4103	从3#Y3 右侧三色灯（红）
M4104	从3#Y4 右侧三色灯（绿）
M4105	从3#Y5 右侧三色灯（黄）
M4106	从3#Y6 出料三色灯（红）
M4107	从3#Y7 出料三色灯（绿）
M4108	从3#Y10 出料三色灯（黄）
M103	从站4#进料皮带速度切换=0 正常，=1低速
M104	从站5#进料皮带速度切换=0 正常，=1低速
M105	从站6#进料皮带速度切换=0 正常，=1低速
M106	从站7#进料皮带速度切换=0 正常，=1低速
M107	从站8#进料皮带速度切换=0 正常，=1低速
M108	从站9#进料皮带速度切换=0 正常，=1低速
M109	从站10#进料皮带速度切换=0 正常，=1低速
M110	从站11#进料皮带速度切换=0 正常，=1低速
M111	从站12#进料皮带速度切换=0 正常，=1低速
M112	从站13#进料皮带速度切换=0 正常，=1低速
M1829	从1出料异常
M1830	从2左侧小车未到位异常
M1831	从2左侧料满异常
M1832	从2左侧出料异常
M1833	从2右侧小车未到位异常
M1834	从2右侧料满异常
M1835	从2右侧出料异常
M1836	从2出料异常
M1837	从3左侧小车未到位异常
M1838	从3左侧料满异常
M1839	从3左侧出料异常
M1840	从3右侧小车未到位异常
M1841	从3右侧料满异常
M1842	从3右侧出料异常
M1843	从3出料异常
M1611	从1已进料
M120	从1#出料
M121	从1#左出料
M122	从1#右出料
T402	从1出料超时
T403	从1左出料超时
T404	从1右出料超时
HD101	从1出料超时